Fanuc KAREL source: CNC_DYN_DISR.kl

PROGRAM T
%NOLOCKGROUP
VAR
 v0 : REAL
 v1 : STRING[40]
 v2 : INTEGER
BEGIN
 CNC_DYN_DISR(v0, v1, v2)
END T
